LIN {X 0,Y 42.172,Z 287.47,A -85,B 0,C 180,E1 -31499.066,E2 -31499.066} C_VEL
LIN {X 0,Y 52.714,Z 280.07,A -85,B 0,C 180,E1 -31500.839,E2 -31500.839} C_VEL
LIN {X 0,Y 63.29,Z 270.881,A -85,B 0,C 180,E1 -31502.039,E2 -31502.039} C_VEL
LIN {X 0,Y 72.989,Z 260.276,A -85,B 0,C 180,E1 -31502.613,E2 -31502.613} C_VEL
LIN {X 0,Y 80.934,Z 249.462,A -85,B 0,C 180,E1 -31503.038,E2 -31503.038} C_VEL
LIN {X 0,Y 87.108,Z 238.971,A -85,B 0,C 180,E1 -31503.228,E2 -31503.228} C_VEL
LIN {X 0,Y 92.563,Z 227.039,A -85,B 0,C 180,E1 -31503.402,E2 -31503.402} C_VEL
LIN {X 0,Y 96.805,Z 214.476,A -85,B 0,C 180,E1 -31503.66,E2 -31503.66} C_VEL
LIN {X 0,Y 98.597,Z 207.38,A -85,B 0,C 180,E1 -31503.833,E2 -31503.833} C_VEL
LIN {X 0,Y 95.469,Z 218.938,A -85,B 0,C 180,E1 -31504.249,E2 -31504.249} C_VEL
LIN {X 0,Y 90.793,Z 231.207,A -85,B 0,C 180,E1 -31504.729,E2 -31504.729} C_VEL
LIN {X 0,Y 84.69,Z 243.28,A -85,B 0,C 180,E1 -31505.259,E2 -31505.259} C_VEL
LIN {X 0,Y 77.709,Z 254.057,A -85,B 0,C 180,E1 -31505.839,E2 -31505.839} C_VEL
LIN {X 0,Y 68.988,Z 264.804,A -85,B 0,C 180,E1 -31506.67,E2 -31506.67} C_VEL
LIN {X 0,Y 60.272,Z 273.542,A -85,B 0,C 180,E1 -31507.647,E2 -31507.647} C_VEL
LIN {X 0,Y 49.845,Z 282.043,A -85,B 0,C 180,E1 -31509.274,E2 -31509.274} C_VEL
LIN {X 0,Y 39.461,Z 288.851,A -85,B 0,C 180,E1 -31511.619,E2 -31511.619} C_VEL
LIN {X 0,Y 29.179,Z 294.298,A -85,B 0,C 180,E1 -31515.557,E2 -31515.557} C_VEL
LIN {X 0,Y 19.097,Z 298.577,A -85,B 0,C 180,E1 -31523.085,E2 -31523.085} C_VEL
LIN {X 0,Y 9.829,Z 301.808,A -85,B 0,C 180,E1 -31544.375,E2 -31544.375} C_VEL
LIN {X 0,Y 6.304,Z 303.878,A -85,B 0,C 180,E1 -31613.698,E2 -31613.698} C_VEL
LIN {X 0,Y 14.631,Z 305.459,A -85,B 0,C 180,E1 -31663.914,E2 -31663.914} C_VEL
LIN {X 0,Y 28.166,Z 305.864,A -85,B 0,C 180,E1 -31676.524,E2 -31676.524} C_VEL
LIN {X 0,Y 32.707,Z 305.617,A -85,B 0,C 180,E1 -31678.423,E2 -31678.423} C_VEL
LIN {X 0,Y 34.772,Z 307.614,A -85,B 0,C 180,E1 -31679.12,E2 -31679.12} C_VEL
LIN {X 0,Y 34.772,Z 600,A -85,B 0,C 180,E1 -31679.12,E2 -31679.12} C_VEL
LIN {X 0,Y 34.772,Z 600,A -85,B 0,C 180,E1 -31679.12,E2 -31679.12}

QRS_NEXT_CUT()

QRS_NEXT()
QRS_HOME()

END
